FUNCTION_BLOCK AnalogLedDisplay010
VAR
	nOutput	AT%Q*	: INT;
END_VAR

PROPERTY DisplayedValue : LREAL
GET
DisplayedValue := F_Scale ( nOutput, 0, 32767, 0, 10 );
END_GET
END_PROPERTY

METHOD SetValue : BOOL
VAR_INPUT
	nValue	: INT;
END_VAR
nOutput := nValue;

SetValue := TRUE;
END_METHOD

END_FUNCTION_BLOCK

(* stored: Version 1.1.0.1
   POU AnalogLedDisplay010: Id {beca59ff-9607-4905-9f5a-6a96fef03655}, SpecialFunc None
   Property DisplayedValue: Id {5300ff47-5ebc-4a5e-8102-f41622631bf5}
   Get Get: Id {1806d3fc-ffc4-44b6-a979-610a4e37d266}
   Method SetValue: Id {bdac92a1-cbc3-4344-b710-6066affbd8c6} *)
